// TIA Portal V17 export
// export: Created 2026-04-12T10:32:02.7096172Z, ExportSetting WithDefaults, DisplayName Totally Integrated Automation Portal, DisplayVersion V17 Update 4, DisplayName TIA Portal Openness, DisplayVersion V17 Update 4, DisplayName TIA Portal Version Control Interface, DisplayVersion V17, DisplayName SINAMICS Startdrive Advanced, DisplayVersion V17, DisplayName SINAMICS Startdrive G130, G150, S120, S150, SINAMICS MV, S210, DisplayVersion V17, DisplayName SINAMICS Startdrive G110M, G120, G120C, G120D, G120P, G115D, DisplayVersion V17, DisplayName STEP 7 Professional, DisplayVersion V17 Update 4, DisplayName STEP 7 Safety, DisplayVersion V17, DisplayName WinCC Advanced, DisplayVersion V17 Update 4
FUNCTION_BLOCK "烧嘴控制"   // FB1, LAD
{ S7_Optimized_Access := 'TRUE' }
VERSION : 0.1
// stored: AutoNumber true, IsIECCheckEnabled false, IsRetainMemResEnabled false, MemoryReserve 100, SetENOAutomatically false, UDAEnableTagReadback false
   VAR_INPUT
      测量值 : Real;
      设定值 : Real;
      小火反馈 : Bool;
      故障反馈 : Bool;
      自动 : Bool;
      手动小火 : Bool;
      手动大火 : Bool;
      PID大火输出 : Bool;
      控温通讯状态 : Bool;
   END_VAR
   VAR_OUTPUT
      小火输出 : Bool;
      大火输出 : Bool;
      复位输出 : Bool;
      自动复位失败 : Bool;
      超温标志 : Bool;
   END_VAR
   VAR
      过程温度 : Real;
      过程温度差值 : Real;
      过程温度差值上限 : Real;
      过程温度差值下限 : Real;
      温度差值 : Real;
      "1秒脉冲1" : Bool;
      复位次数脉冲 : Bool;
      复位定时器1 : IEC_TIMER;
      复位定时器2 { S7_SetPoint := 'True'} : IEC_TIMER;
      趋势定时器 { S7_SetPoint := 'True'} : IEC_TIMER;
      小火定时器 { S7_SetPoint := 'True'} : IEC_TIMER;
      小火保持定时器 { S7_SetPoint := 'True'} : IEC_TIMER;
      复位脉冲 { S7_SetPoint := 'True'} : Bool;
      复位次数 : Int;
      趋势定时器脉冲1 : Bool;
      趋势定时器脉冲2 : Bool;
      趋势定时器复位 : Bool;
      温度上升趋势 : Bool;
      温度下降趋势 : Bool;
      大火设定时间 : Int;
      大火运行时间 : Int;
      内部自动大火输出 : Bool;
      "1秒脉冲" { S7_SetPoint := 'True'} : Bool;
      小火保持标志 : Bool;
      小火保持脉冲 : Bool;
      小火保持取消脉冲1 : Bool;
      小火保持取消脉冲2 : Bool;
   END_VAR
   VAR_TEMP   // added for the SCL form of the ladder/FBD networks
      _w1 : Bool;
      _w2 : Bool;
      _w3 : Bool;
      _w4 : Bool;
      _w5 : Bool;
      _w6 : Bool;
      _w7 : Bool;
   END_VAR
BEGIN

REGION Network 1: 温度差值，超温标志
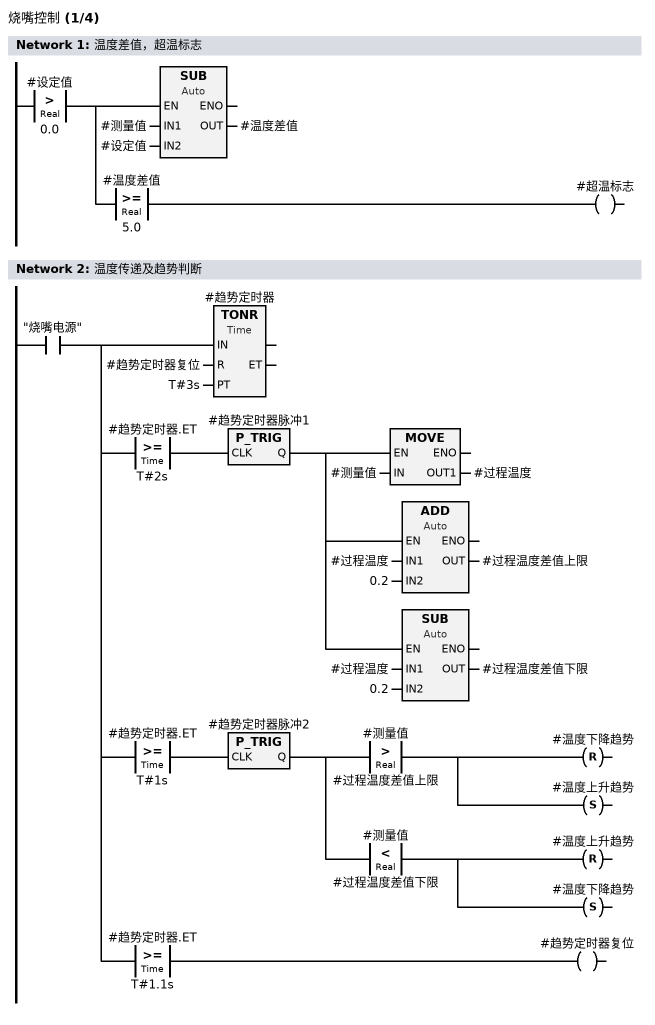
   RUNG wire#powerrail
      { S7_Templates := "SrcType := Real" } GT_Contact(in1 := #设定值, in2 := 0.0)
      wire#w1
      Sub(in1 := #测量值, in2 := #设定值, out => #温度差值)
   END_RUNG
   RUNG wire#w1
      { S7_Templates := "SrcType := Real" } GE_Contact(in1 := #温度差值, in2 := 5.0)
      Coil( #超温标志 )
   END_RUNG
   // the same network as SCL:
   #_w1 := #设定值 > 0.0;
   IF #_w1 THEN #温度差值 := #测量值 - #设定值; END_IF;
   #超温标志 := #_w1 AND (#温度差值 >= 5.0);
END_REGION

REGION Network 2: 温度传递及趋势判断
   RUNG wire#powerrail
      Contact( "烧嘴电源" )
      wire#w1
      { S7_Templates := "time_type := Time" } #趋势定时器.TONR(r := #趋势定时器复位, pt := T#3s, et =>)
   END_RUNG
   RUNG wire#w1
      { S7_Templates := "SrcType := Time" } GE_Contact(in1 := #趋势定时器.ET, in2 := T#2s)
      P_Trig( #趋势定时器脉冲1 )
      wire#w2
      Move(in := #测量值, out1 => #过程温度)
   END_RUNG
   RUNG wire#w2
      Add(in1 := #过程温度, in2 := 0.2, out => #过程温度差值上限)
   END_RUNG
   RUNG wire#w2
      Sub(in1 := #过程温度, in2 := 0.2, out => #过程温度差值下限)
   END_RUNG
   RUNG wire#w1
      { S7_Templates := "SrcType := Time" } GE_Contact(in1 := #趋势定时器.ET, in2 := T#1s)
      P_Trig( #趋势定时器脉冲2 )
      wire#w3
      { S7_Templates := "SrcType := Real" } GT_Contact(in1 := #测量值, in2 := #过程温度差值上限)
      wire#w4
      R_Coil( #温度下降趋势 )
   END_RUNG
   RUNG wire#w4
      S_Coil( #温度上升趋势 )
   END_RUNG
   RUNG wire#w3
      { S7_Templates := "SrcType := Real" } LT_Contact(in1 := #测量值, in2 := #过程温度差值下限)
      wire#w5
      R_Coil( #温度上升趋势 )
   END_RUNG
   RUNG wire#w5
      S_Coil( #温度下降趋势 )
   END_RUNG
   RUNG wire#w1
      { S7_Templates := "SrcType := Time" } GE_Contact(in1 := #趋势定时器.ET, in2 := T#1.1s)
      Coil( #趋势定时器复位 )
   END_RUNG
   // the same network as SCL:
   #趋势定时器.TONR(IN := "烧嘴电源", R := #趋势定时器复位, PT := T#3s);
   #_w1 := "烧嘴电源" AND (#趋势定时器.ET >= T#2s);
   #_w2 := #_w1 AND NOT #趋势定时器脉冲1;   // rising edge
   #趋势定时器脉冲1 := #_w1;
   IF #_w2 THEN
       #过程温度 := #测量值;
       #过程温度差值上限 := #过程温度 + 0.2;
       #过程温度差值下限 := #过程温度 - 0.2;
   END_IF;
   #_w3 := "烧嘴电源" AND (#趋势定时器.ET >= T#1s);
   #_w4 := #_w3 AND NOT #趋势定时器脉冲2;   // rising edge
   #趋势定时器脉冲2 := #_w3;
   IF #_w4 AND (#测量值 > #过程温度差值上限) THEN
       #温度下降趋势 := FALSE;
       #温度上升趋势 := TRUE;
   END_IF;
   IF #_w4 AND (#测量值 < #过程温度差值下限) THEN
       #温度上升趋势 := FALSE;
       #温度下降趋势 := TRUE;
   END_IF;
   #趋势定时器复位 := "烧嘴电源" AND (#趋势定时器.ET >= T#1.1s);
END_REGION

REGION Network 3: 点火
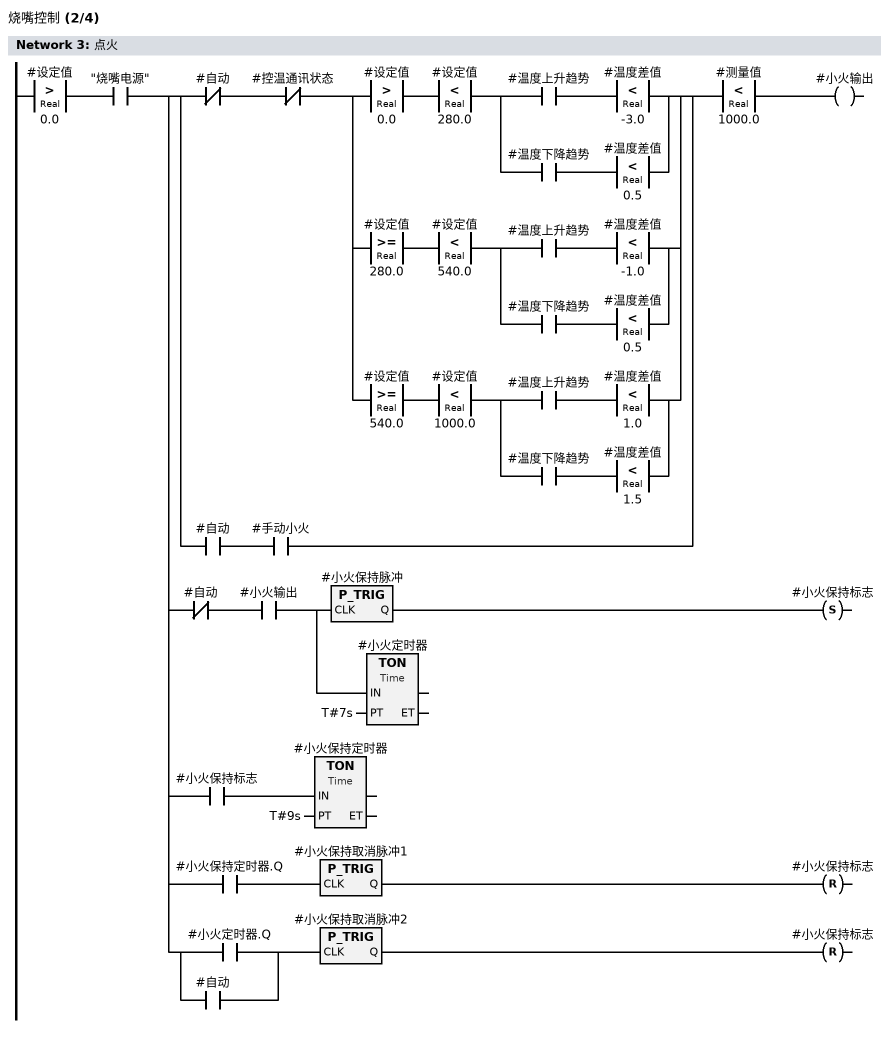
   RUNG wire#powerrail
      { S7_Templates := "SrcType := Real" } GT_Contact(in1 := #设定值, in2 := 0.0)
      Contact( "烧嘴电源" )
      wire#w1
      I_Contact( #自动 )
      I_Contact( #控温通讯状态 )
      wire#w2
      { S7_Templates := "SrcType := Real" } GT_Contact(in1 := #设定值, in2 := 0.0)
      { S7_Templates := "SrcType := Real" } LT_Contact(in1 := #设定值, in2 := 280.0)
      wire#w3
      Contact( #温度上升趋势 )
      { S7_Templates := "SrcType := Real" } LT_Contact(in1 := #温度差值, in2 := -3.0)
      wire#w4
      { S7_Templates := "SrcType := Real" } LT_Contact(in1 := #测量值, in2 := 1000.0)
      Coil( #小火输出 )
   END_RUNG
   RUNG wire#w3
      Contact( #温度下降趋势 )
      { S7_Templates := "SrcType := Real" } LT_Contact(in1 := #温度差值, in2 := 0.5)
   END_RUNG wire#w4
   RUNG wire#w2
      { S7_Templates := "SrcType := Real" } GE_Contact(in1 := #设定值, in2 := 280.0)
      { S7_Templates := "SrcType := Real" } LT_Contact(in1 := #设定值, in2 := 540.0)
      wire#w5
      Contact( #温度上升趋势 )
      { S7_Templates := "SrcType := Real" } LT_Contact(in1 := #温度差值, in2 := -1.0)
   END_RUNG wire#w4
   RUNG wire#w5
      Contact( #温度下降趋势 )
      { S7_Templates := "SrcType := Real" } LT_Contact(in1 := #温度差值, in2 := 0.5)
   END_RUNG wire#w4
   RUNG wire#w2
      { S7_Templates := "SrcType := Real" } GE_Contact(in1 := #设定值, in2 := 540.0)
      { S7_Templates := "SrcType := Real" } LT_Contact(in1 := #设定值, in2 := 1000.0)
      wire#w6
      Contact( #温度上升趋势 )
      { S7_Templates := "SrcType := Real" } LT_Contact(in1 := #温度差值, in2 := 1.0)
   END_RUNG wire#w4
   RUNG wire#w6
      Contact( #温度下降趋势 )
      { S7_Templates := "SrcType := Real" } LT_Contact(in1 := #温度差值, in2 := 1.5)
   END_RUNG wire#w4
   RUNG wire#w1
      Contact( #自动 )
      Contact( #手动小火 )
   END_RUNG wire#w4
   RUNG wire#w1
      I_Contact( #自动 )
      Contact( #小火输出 )
      wire#w7
      P_Trig( #小火保持脉冲 )
      S_Coil( #小火保持标志 )
   END_RUNG
   RUNG wire#w7
      { S7_Templates := "time_type := Time" } #小火定时器.TON(pt := T#7s, et =>)
   END_RUNG
   RUNG wire#w1
      Contact( #小火保持标志 )
      { S7_Templates := "time_type := Time" } #小火保持定时器.TON(pt := T#9s, et =>)
   END_RUNG
   RUNG wire#w1
      Contact( #小火保持定时器.Q )
      P_Trig( #小火保持取消脉冲1 )
      R_Coil( #小火保持标志 )
   END_RUNG
   RUNG wire#w1
      Contact( #小火定时器.Q )
      wire#w8
      P_Trig( #小火保持取消脉冲2 )
      R_Coil( #小火保持标志 )
   END_RUNG
   RUNG wire#w1
      Contact( #自动 )
   END_RUNG wire#w8
   // the same network as SCL:
   #_w1 := (#设定值 > 0.0) AND "烧嘴电源";
   #小火输出 := #_w1 AND ((NOT #自动 AND NOT #控温通讯状态 AND (((#设定值 > 0.0) AND (#设定值 < 280.0) AND ((#温度上升趋势 AND (#温度差值 < (-3.0))) OR (#温度下降趋势 AND (#温度差值 < 0.5)))) OR ((#设定值 >= 280.0) AND (#设定值 < 540.0) AND ((#温度上升趋势 AND (#温度差值 < (-1.0))) OR (#温度下降趋势 AND (#温度差值 < 0.5)))) OR ((#设定值 >= 540.0) AND (#设定值 < 1000.0) AND ((#温度上升趋势 AND (#温度差值 < 1.0)) OR (#温度下降趋势 AND (#温度差值 < 1.5)))))) OR (#自动 AND #手动小火)) AND (#测量值 < 1000.0);
   #_w2 := #_w1 AND NOT #自动 AND #小火输出;
   #_w3 := #_w2 AND NOT #小火保持脉冲;   // rising edge
   #小火保持脉冲 := #_w2;
   IF #_w3 THEN #小火保持标志 := TRUE; END_IF;
   #小火定时器.TON(IN := #_w2, PT := T#7s);
   #小火保持定时器.TON(IN := #_w1 AND #小火保持标志, PT := T#9s);
   #_w4 := #_w1 AND #小火保持定时器.Q;
   #_w5 := #_w4 AND NOT #小火保持取消脉冲1;   // rising edge
   #小火保持取消脉冲1 := #_w4;
   IF #_w5 THEN #小火保持标志 := FALSE; END_IF;
   #_w6 := #_w1 AND (#小火定时器.Q OR #自动);
   #_w7 := #_w6 AND NOT #小火保持取消脉冲2;   // rising edge
   #小火保持取消脉冲2 := #_w6;
   IF #_w7 THEN #小火保持标志 := FALSE; END_IF;
END_REGION

REGION Network 4: 大火时间设定
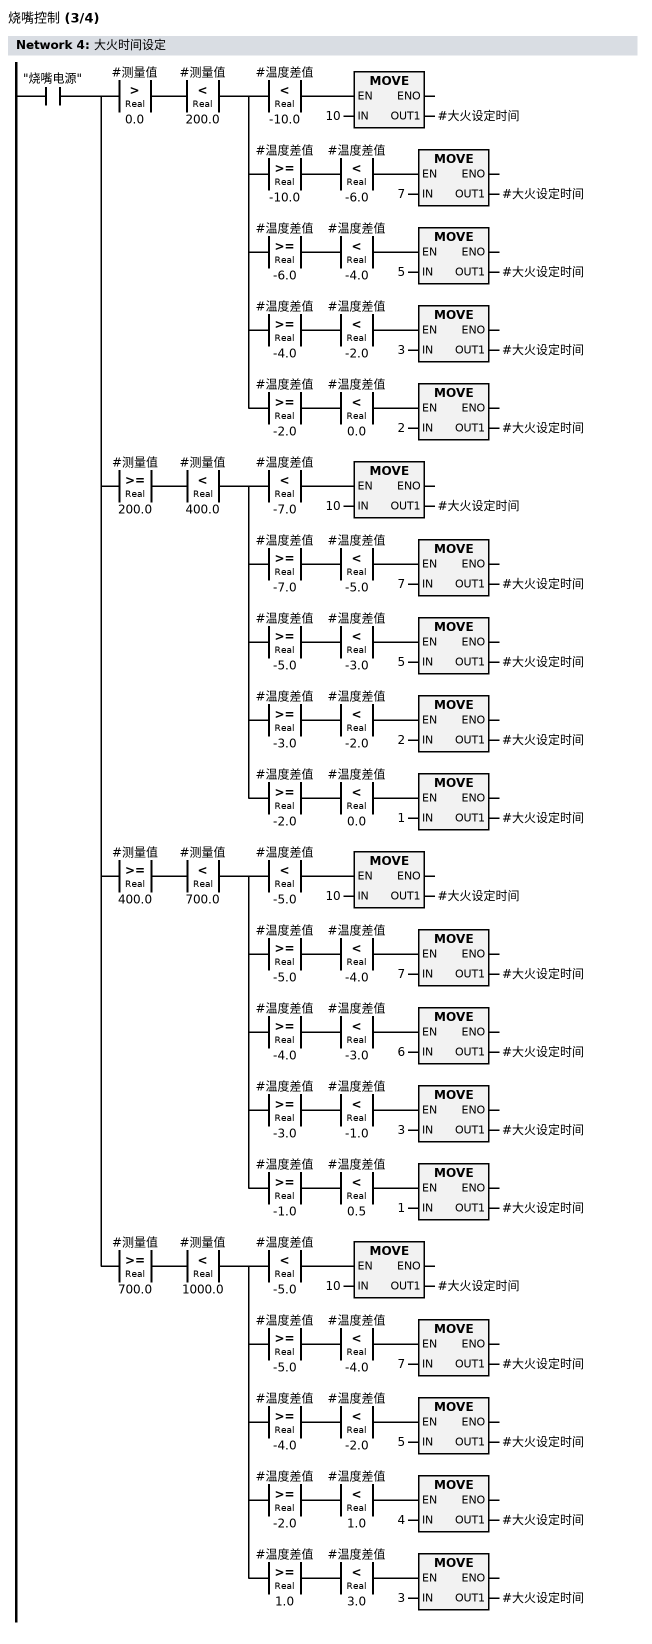
   RUNG wire#powerrail
      Contact( "烧嘴电源" )
      wire#w1
      { S7_Templates := "SrcType := Real" } GT_Contact(in1 := #测量值, in2 := 0.0)
      { S7_Templates := "SrcType := Real" } LT_Contact(in1 := #测量值, in2 := 200.0)
      wire#w2
      { S7_Templates := "SrcType := Real" } LT_Contact(in1 := #温度差值, in2 := -10.0)
      Move(in := 10, out1 => #大火设定时间)
   END_RUNG
   RUNG wire#w2
      { S7_Templates := "SrcType := Real" } GE_Contact(in1 := #温度差值, in2 := -10.0)
      { S7_Templates := "SrcType := Real" } LT_Contact(in1 := #温度差值, in2 := -6.0)
      Move(in := 7, out1 => #大火设定时间)
   END_RUNG
   RUNG wire#w2
      { S7_Templates := "SrcType := Real" } GE_Contact(in1 := #温度差值, in2 := -6.0)
      { S7_Templates := "SrcType := Real" } LT_Contact(in1 := #温度差值, in2 := -4.0)
      Move(in := 5, out1 => #大火设定时间)
   END_RUNG
   RUNG wire#w2
      { S7_Templates := "SrcType := Real" } GE_Contact(in1 := #温度差值, in2 := -4.0)
      { S7_Templates := "SrcType := Real" } LT_Contact(in1 := #温度差值, in2 := -2.0)
      Move(in := 3, out1 => #大火设定时间)
   END_RUNG
   RUNG wire#w2
      { S7_Templates := "SrcType := Real" } GE_Contact(in1 := #温度差值, in2 := -2.0)
      { S7_Templates := "SrcType := Real" } LT_Contact(in1 := #温度差值, in2 := 0.0)
      Move(in := 2, out1 => #大火设定时间)
   END_RUNG
   RUNG wire#w1
      { S7_Templates := "SrcType := Real" } GE_Contact(in1 := #测量值, in2 := 200.0)
      { S7_Templates := "SrcType := Real" } LT_Contact(in1 := #测量值, in2 := 400.0)
      wire#w3
      { S7_Templates := "SrcType := Real" } LT_Contact(in1 := #温度差值, in2 := -7.0)
      Move(in := 10, out1 => #大火设定时间)
   END_RUNG
   RUNG wire#w3
      { S7_Templates := "SrcType := Real" } GE_Contact(in1 := #温度差值, in2 := -7.0)
      { S7_Templates := "SrcType := Real" } LT_Contact(in1 := #温度差值, in2 := -5.0)
      Move(in := 7, out1 => #大火设定时间)
   END_RUNG
   RUNG wire#w3
      { S7_Templates := "SrcType := Real" } GE_Contact(in1 := #温度差值, in2 := -5.0)
      { S7_Templates := "SrcType := Real" } LT_Contact(in1 := #温度差值, in2 := -3.0)
      Move(in := 5, out1 => #大火设定时间)
   END_RUNG
   RUNG wire#w3
      { S7_Templates := "SrcType := Real" } GE_Contact(in1 := #温度差值, in2 := -3.0)
      { S7_Templates := "SrcType := Real" } LT_Contact(in1 := #温度差值, in2 := -2.0)
      Move(in := 2, out1 => #大火设定时间)
   END_RUNG
   RUNG wire#w3
      { S7_Templates := "SrcType := Real" } GE_Contact(in1 := #温度差值, in2 := -2.0)
      { S7_Templates := "SrcType := Real" } LT_Contact(in1 := #温度差值, in2 := 0.0)
      Move(in := 1, out1 => #大火设定时间)
   END_RUNG
   RUNG wire#w1
      { S7_Templates := "SrcType := Real" } GE_Contact(in1 := #测量值, in2 := 400.0)
      { S7_Templates := "SrcType := Real" } LT_Contact(in1 := #测量值, in2 := 700.0)
      wire#w4
      { S7_Templates := "SrcType := Real" } LT_Contact(in1 := #温度差值, in2 := -5.0)
      Move(in := 10, out1 => #大火设定时间)
   END_RUNG
   RUNG wire#w4
      { S7_Templates := "SrcType := Real" } GE_Contact(in1 := #温度差值, in2 := -5.0)
      { S7_Templates := "SrcType := Real" } LT_Contact(in1 := #温度差值, in2 := -4.0)
      Move(in := 7, out1 => #大火设定时间)
   END_RUNG
   RUNG wire#w4
      { S7_Templates := "SrcType := Real" } GE_Contact(in1 := #温度差值, in2 := -4.0)
      { S7_Templates := "SrcType := Real" } LT_Contact(in1 := #温度差值, in2 := -3.0)
      Move(in := 6, out1 => #大火设定时间)
   END_RUNG
   RUNG wire#w4
      { S7_Templates := "SrcType := Real" } GE_Contact(in1 := #温度差值, in2 := -3.0)
      { S7_Templates := "SrcType := Real" } LT_Contact(in1 := #温度差值, in2 := -1.0)
      Move(in := 3, out1 => #大火设定时间)
   END_RUNG
   RUNG wire#w4
      { S7_Templates := "SrcType := Real" } GE_Contact(in1 := #温度差值, in2 := -1.0)
      { S7_Templates := "SrcType := Real" } LT_Contact(in1 := #温度差值, in2 := 0.5)
      Move(in := 1, out1 => #大火设定时间)
   END_RUNG
   RUNG wire#w1
      { S7_Templates := "SrcType := Real" } GE_Contact(in1 := #测量值, in2 := 700.0)
      { S7_Templates := "SrcType := Real" } LT_Contact(in1 := #测量值, in2 := 1000.0)
      wire#w5
      { S7_Templates := "SrcType := Real" } LT_Contact(in1 := #温度差值, in2 := -5.0)
      Move(in := 10, out1 => #大火设定时间)
   END_RUNG
   RUNG wire#w5
      { S7_Templates := "SrcType := Real" } GE_Contact(in1 := #温度差值, in2 := -5.0)
      { S7_Templates := "SrcType := Real" } LT_Contact(in1 := #温度差值, in2 := -4.0)
      Move(in := 7, out1 => #大火设定时间)
   END_RUNG
   RUNG wire#w5
      { S7_Templates := "SrcType := Real" } GE_Contact(in1 := #温度差值, in2 := -4.0)
      { S7_Templates := "SrcType := Real" } LT_Contact(in1 := #温度差值, in2 := -2.0)
      Move(in := 5, out1 => #大火设定时间)
   END_RUNG
   RUNG wire#w5
      { S7_Templates := "SrcType := Real" } GE_Contact(in1 := #温度差值, in2 := -2.0)
      { S7_Templates := "SrcType := Real" } LT_Contact(in1 := #温度差值, in2 := 1.0)
      Move(in := 4, out1 => #大火设定时间)
   END_RUNG
   RUNG wire#w5
      { S7_Templates := "SrcType := Real" } GE_Contact(in1 := #温度差值, in2 := 1.0)
      { S7_Templates := "SrcType := Real" } LT_Contact(in1 := #温度差值, in2 := 3.0)
      Move(in := 3, out1 => #大火设定时间)
   END_RUNG
   // the same network as SCL:
   #_w1 := "烧嘴电源" AND (#测量值 > 0.0) AND (#测量值 < 200.0);
   IF #_w1 AND (#温度差值 < (-10.0)) THEN #大火设定时间 := 10; END_IF;
   IF #_w1 AND (#温度差值 >= (-10.0)) AND (#温度差值 < (-6.0)) THEN #大火设定时间 := 7; END_IF;
   IF #_w1 AND (#温度差值 >= (-6.0)) AND (#温度差值 < (-4.0)) THEN #大火设定时间 := 5; END_IF;
   IF #_w1 AND (#温度差值 >= (-4.0)) AND (#温度差值 < (-2.0)) THEN #大火设定时间 := 3; END_IF;
   IF #_w1 AND (#温度差值 >= (-2.0)) AND (#温度差值 < 0.0) THEN #大火设定时间 := 2; END_IF;
   #_w2 := "烧嘴电源" AND (#测量值 >= 200.0) AND (#测量值 < 400.0);
   IF #_w2 AND (#温度差值 < (-7.0)) THEN #大火设定时间 := 10; END_IF;
   IF #_w2 AND (#温度差值 >= (-7.0)) AND (#温度差值 < (-5.0)) THEN #大火设定时间 := 7; END_IF;
   IF #_w2 AND (#温度差值 >= (-5.0)) AND (#温度差值 < (-3.0)) THEN #大火设定时间 := 5; END_IF;
   IF #_w2 AND (#温度差值 >= (-3.0)) AND (#温度差值 < (-2.0)) THEN #大火设定时间 := 2; END_IF;
   IF #_w2 AND (#温度差值 >= (-2.0)) AND (#温度差值 < 0.0) THEN #大火设定时间 := 1; END_IF;
   #_w3 := "烧嘴电源" AND (#测量值 >= 400.0) AND (#测量值 < 700.0);
   IF #_w3 AND (#温度差值 < (-5.0)) THEN #大火设定时间 := 10; END_IF;
   IF #_w3 AND (#温度差值 >= (-5.0)) AND (#温度差值 < (-4.0)) THEN #大火设定时间 := 7; END_IF;
   IF #_w3 AND (#温度差值 >= (-4.0)) AND (#温度差值 < (-3.0)) THEN #大火设定时间 := 6; END_IF;
   IF #_w3 AND (#温度差值 >= (-3.0)) AND (#温度差值 < (-1.0)) THEN #大火设定时间 := 3; END_IF;
   IF #_w3 AND (#温度差值 >= (-1.0)) AND (#温度差值 < 0.5) THEN #大火设定时间 := 1; END_IF;
   #_w4 := "烧嘴电源" AND (#测量值 >= 700.0) AND (#测量值 < 1000.0);
   IF #_w4 AND (#温度差值 < (-5.0)) THEN #大火设定时间 := 10; END_IF;
   IF #_w4 AND (#温度差值 >= (-5.0)) AND (#温度差值 < (-4.0)) THEN #大火设定时间 := 7; END_IF;
   IF #_w4 AND (#温度差值 >= (-4.0)) AND (#温度差值 < (-2.0)) THEN #大火设定时间 := 5; END_IF;
   IF #_w4 AND (#温度差值 >= (-2.0)) AND (#温度差值 < 1.0) THEN #大火设定时间 := 4; END_IF;
   IF #_w4 AND (#温度差值 >= 1.0) AND (#温度差值 < 3.0) THEN #大火设定时间 := 3; END_IF;
END_REGION

REGION Network 5: 大火运行计时
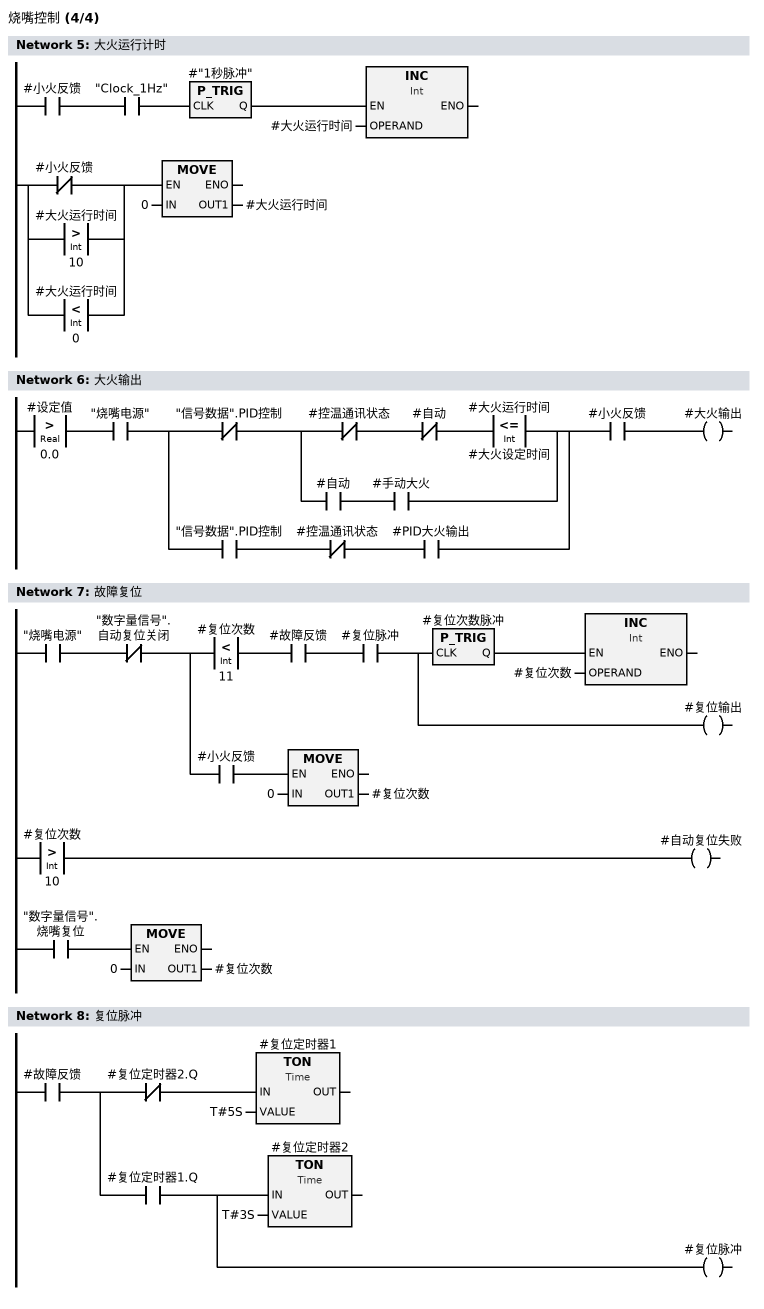
   RUNG wire#powerrail
      Contact( #小火反馈 )
      Contact( "Clock_1Hz" )
      P_Trig( #"1秒脉冲" )
      { S7_Templates := "DestType := Int" } Inc( #大火运行时间 )
   END_RUNG
   RUNG wire#powerrail
      I_Contact( #小火反馈 )
      wire#w1
      Move(in := 0, out1 => #大火运行时间)
   END_RUNG
   RUNG wire#powerrail
      { S7_Templates := "SrcType := Int" } GT_Contact(in1 := #大火运行时间, in2 := 10)
   END_RUNG wire#w1
   RUNG wire#powerrail
      { S7_Templates := "SrcType := Int" } LT_Contact(in1 := #大火运行时间, in2 := 0)
   END_RUNG wire#w1
   // the same network as SCL:
   #_w1 := #小火反馈 AND "Clock_1Hz";
   #_w2 := #_w1 AND NOT #"1秒脉冲";   // rising edge
   #"1秒脉冲" := #_w1;
   IF #_w2 THEN #大火运行时间 := #大火运行时间 + 1; END_IF;
   IF NOT #小火反馈 OR (#大火运行时间 > 10) OR (#大火运行时间 < 0) THEN #大火运行时间 := 0; END_IF;
END_REGION

REGION Network 6: 大火输出
   RUNG wire#powerrail
      { S7_Templates := "SrcType := Real" } GT_Contact(in1 := #设定值, in2 := 0.0)
      Contact( "烧嘴电源" )
      wire#w1
      I_Contact( "信号数据".PID控制 )
      wire#w2
      I_Contact( #控温通讯状态 )
      I_Contact( #自动 )
      { S7_Templates := "SrcType := Int" } LE_Contact(in1 := #大火运行时间, in2 := #大火设定时间)
      wire#w3
      Contact( #小火反馈 )
      Coil( #大火输出 )
   END_RUNG
   RUNG wire#w2
      Contact( #自动 )
      Contact( #手动大火 )
   END_RUNG wire#w3
   RUNG wire#w1
      Contact( "信号数据".PID控制 )
      I_Contact( #控温通讯状态 )
      Contact( #PID大火输出 )
   END_RUNG wire#w3
   // the same network as SCL:
   #大火输出 := (#设定值 > 0.0) AND "烧嘴电源" AND ((NOT "信号数据".PID控制 AND ((NOT #控温通讯状态 AND NOT #自动 AND (#大火运行时间 <= #大火设定时间)) OR (#自动 AND #手动大火))) OR ("信号数据".PID控制 AND NOT #控温通讯状态 AND #PID大火输出)) AND #小火反馈;
END_REGION

REGION Network 7: 故障复位
   RUNG wire#powerrail
      Contact( "烧嘴电源" )
      I_Contact( "数字量信号".自动复位关闭 )
      wire#w1
      { S7_Templates := "SrcType := Int" } LT_Contact(in1 := #复位次数, in2 := 11)
      Contact( #故障反馈 )
      Contact( #复位脉冲 )
      wire#w2
      P_Trig( #复位次数脉冲 )
      { S7_Templates := "DestType := Int" } Inc( #复位次数 )
   END_RUNG
   RUNG wire#w2
      Coil( #复位输出 )
   END_RUNG
   RUNG wire#w1
      Contact( #小火反馈 )
      Move(in := 0, out1 => #复位次数)
   END_RUNG
   RUNG wire#powerrail
      { S7_Templates := "SrcType := Int" } GT_Contact(in1 := #复位次数, in2 := 10)
      Coil( #自动复位失败 )
   END_RUNG
   RUNG wire#powerrail
      Contact( "数字量信号".烧嘴复位 )
      Move(in := 0, out1 => #复位次数)
   END_RUNG
   // the same network as SCL:
   #_w1 := "烧嘴电源" AND NOT "数字量信号".自动复位关闭;
   #_w2 := #_w1 AND (#复位次数 < 11) AND #故障反馈 AND #复位脉冲;
   #_w3 := #_w2 AND NOT #复位次数脉冲;   // rising edge
   #复位次数脉冲 := #_w2;
   IF #_w3 THEN #复位次数 := #复位次数 + 1; END_IF;
   #复位输出 := #_w2;
   IF #_w1 AND #小火反馈 THEN #复位次数 := 0; END_IF;
   #自动复位失败 := #复位次数 > 10;
   IF "数字量信号".烧嘴复位 THEN #复位次数 := 0; END_IF;
END_REGION

REGION Network 8: 复位脉冲
   #复位定时器1.TON(IN := #故障反馈 AND NOT #复位定时器2.Q, PT := T#5S);   // TON coil
   #_w1 := #故障反馈 AND #复位定时器1.Q;
   #复位定时器2.TON(IN := #_w1, PT := T#3S);   // TON coil
   #复位脉冲 := #_w1;
END_REGION
END_FUNCTION_BLOCK
